Universal Robots PolyScope program: 20241121_contact_test1.urp

Program 20241121_contact_test1 (installation=20240827 directory=/programs/Demos/contact_test createdIn=5.15.1 lastSavedIn=5.15.1 robotSerialNumber=20245500285)
Calibrated DH parameters: a=[0.000097, -0.210459, -0.026602, 0.000137, 0.000078, 0]; d=[0.162601, 254.180657, -54.076236, -199.970743, 0.099615, 0.099684]; alpha=[1.569796, -0.001455, 0.001957, 1.570525, -1.571561, 0]; deltaTheta=[0, -1.053331, 8.839472, -1.50296, 0.000002, 0]
InitVariablesNode
Robot Program (runOnlyOnce=false)
  Script: usb = rpc_factory("xmlrpc","http://192.168.1.3:9120/RPC2")
  Script: usb.disEnableSlipDetector()
  Popup Message (haltProgram=false message=place check everything is ok! inputType=Text)
  Script: write_output_integer_register(0,1)
  SuppressedNode
    Wait DigitalInput pin=digital_in[0]; digitalValue=1
  SuppressedNode
    MoveJ speed 60 deg/s, acceleration 80 deg/s^2 (useActiveTCP=true) feature=Base
      Waypoint home: TCP in base x=278.361 y=-491.587 z=269.715 mm, rx=-2.164 ry=-2.1556 rz=-0.0005 rad; joints [106.983, -78.785, 80.375, -87.202, -92.296, 107.473] deg; TCP offset x=-0.17 y=0 z=192.95 mm, rx=0 ry=0 rz=0 rad
  Script: usb.open()
  Popup Message (haltProgram=false message=close inputType=Text)
  Script: usb.adaptiveClose()
  SuppressedNode
    Script: usb.enableSlipDetector()
  Wait Sleep waitTime=2
  SuppressedNode
    Halt
  Script: usb.enableSlipDetector()
  Loop Forever
    SuppressedNode
      MoveL speed 100 mm/s, acceleration 500 mm/s^2 (useActiveTCP=true) feature=Base
        Waypoint 路点_1: TCP in base x=278.354 y=-491.58 z=76.094 mm, rx=-2.2854 ry=-2.1556 rz=0 rad; joints [105.754, -74.454, 105.742, -121.331, -90.051, 109.278] deg
          Until EXPRESSION (allowActions=false deceleration=35) ExpressionBranch=tmp[0]>1
        Wait Sleep waitTime=2
        Script: usb.disEnableSlipDetector()
        Waypoint 路点_2: TCP in base x=278.344 y=-491.573 z=202.918 mm, rx=-2.2854 ry=-2.1555 rz=0 rad; joints [105.755, -80.97, 93.805, -102.875, -90.011, 109.282] deg
Thread Thread_1 (runOnlyOnce=false)
  tmp := p[0,0,0,0,0,0]
  Loop Forever
    watchdog := read_input_integer_register(0)
    Script file /programs/pose_register.script
      | tmp[0]=read_input_float_register(0)
      | tmp[1]=read_input_float_register(1)
      | tmp[2]=read_input_float_register(2)
      | tmp[3]=read_input_float_register(3)
      | tmp[4]=read_input_float_register(4)
      | tmp[5]=read_input_float_register(5)
    Script: sync()
